FUNCTION_BLOCK FB_Axis
VAR_OUTPUT
	bError			:	BOOL;				//Error signal
	nErrorID		:	UDINT;				//Error ID
	bMoving			:	BOOL;				// Status of moving
END_VAR
VAR
	bResetDone		:	BOOL;				// Status of function block MC_Reset
	bHaltDone		:	BOOL;				// Status of function block MC_Halt

	bStatusEnable	:	BOOL;				// Enable feedback
	
	fVelocity		:	LREAL;				// Target velocity
	fOverride		:	LREAL := 100;		// Override 100%
	
	fbTriggerHalt	:	R_TRIG;				// Trigger to recognize rising edge of halt input
	fbTriggerReset	:	R_TRIG;				// Trigger to recognize rising edge of reset input
	
	AxisRef			:	AXIS_REF;			// Axis reference (process data plc/nc)
	
	//=============== Motion function blocks =====================
	fbMcPower		:	MC_Power;			// FB for enable and override
	fbMcReset		:	MC_Reset;			// FB to reset axis (errors)
	fbMcStop		:	MC_Stop;				// FB to stop axis
	fbMcHalt		:	MC_Halt;				// FB to halt axis
	fbMcMove		:	Mc_MoveVelocity;	// FB to move axis (velocity movement)
	fbMcMoveAbsolute :	Mc_MoveAbsolute;	// FB to move axis (absolute position)
END_VAR

PROPERTY bState_Enable : BOOL
GET
bState_Enable := bStatusEnable;
END_GET
END_PROPERTY

PROPERTY bState_HaltDone : BOOL
GET
bState_HaltDone := bHaltDone;
END_GET
END_PROPERTY

PROPERTY bState_ResetDone : BOOL
GET
bState_ResetDone := bResetDone;
END_GET
END_PROPERTY

METHOD Enable
VAR_INPUT
	bEnable		:		BOOL;
END_VAR
fbMcPower(	Axis 			:= THIS^.AxisRef,
			Enable 			:=  bEnable,
			Enable_Positive := bEnable,
			Enable_Negative := bEnable,
			Override 		:= THIS^.fOverride,
			Status 			=> THIS^.bStatusEnable);
			
IF fbMcPower.Error THEN
	bError		:= TRUE;
	nErrorID	:= fbMcPower.ErrorID;
END_IF

AxisRef.ReadStatus();		// Axis internal method to read its status

THIS^.bMoving := AxisRef.Status.Moving;
END_METHOD

PROPERTY fTargetVelocity : LREAL
GET
fTargetVelocity := fVelocity;
END_GET
SET
fVelocity := fTargetVelocity;
END_SET
END_PROPERTY

METHOD Halt
VAR_INPUT
	bDriveHalt	:	BOOL;
END_VAR
// Move axis command set to FALSE
IF bDriveHalt THEN
	THIS^.fbMcMove( Axis 				:= THIS^.AxisRef,
					Execute 			:= FALSE);
	// ?? Move Absolute Execute FALSE ??
	THIS^.fbMcMoveAbsolute( Axis 		:= THIS^.AxisRef,
							Execute 	:= FALSE);		
ELSE
	THIS^.bHaltDone := FALSE;				
END_IF

//Trigger
THIS^.fbTriggerHalt(CLK := bDriveHalt);

IF THIS^.fbTriggerHalt.Q THEN
	THIS^.fbMcHalt( Axis			:= THIS^.AxisRef,
					Execute			:= TRUE);
ELSE
	THIS^.fbMcHalt( Axis			:= THIS^.AxisRef);
END_IF

// Done / Error / Aborted
IF THIS^.fbMcHalt.Done OR THIS^.fbMcHalt.Error OR THIS^.fbMcHalt.CommandAborted THEN
	THIS^.bError		:= THIS^.fbMcHalt.Error;
	THIS^.nErrorID		:= THIS^.fbMcHalt.ErrorID;
	THIS^.bHaltDone		:= THIS^.fbMcHalt.Done;

	THIS^.fbMcHalt( Axis 		:= THIS^.AxisRef,
					Execute		:= FALSE);
END_IF
END_METHOD

METHOD MoveBw
VAR_INPUT
END_VAR
IF NOT THIS^.fbMcMove.Error THEN
	fbMcMove(	Axis		:= THIS^.AxisRef,
				Execute		:= TRUE,
				Direction	:= MC_Negative_Direction,
				Velocity	:= THIS^.fVelocity);
END_IF

// Error / Command aborted
IF THIS^.fbMcMove.Error OR THIS^.fbMcMove.CommandAborted THEN
	THIS^.bError			:= THIS^.fbMcMove.Error;
	THIS^.nErrorID			:= THIS^.fbMcMove.ErrorID;
END_IF

	fbMcMove(	Axis		:= THIS^.AxisRef,
				Execute		:= FALSE);
END_METHOD

METHOD MoveFw
VAR_INPUT
END_VAR
IF NOT THIS^.fbMcMove.Error THEN
	fbMcMove(	Axis		:= THIS^.AxisRef,
				Execute		:= TRUE,
				Direction	:= MC_Positive_Direction,
				Velocity	:= THIS^.fVelocity);
END_IF

// Error / Command aborted
IF THIS^.fbMcMove.Error OR THIS^.fbMcMove.CommandAborted THEN
	THIS^.bError			:= THIS^.fbMcMove.Error;
	THIS^.nErrorID			:= THIS^.fbMcMove.ErrorID;
END_IF

	fbMcMove(	Axis		:= THIS^.AxisRef,
				Execute		:= FALSE);
END_METHOD

METHOD Reset
VAR_INPUT
	bDriveReset		:	BOOL;	// Request reset
END_VAR
IF NOT bDriveReset THEN
	THIS^.bResetDone := FALSE;
END_IF

// Trigger
THIS^.fbTriggerReset(CLK 		:= bDriveReset);

IF THIS^.fbTriggerReset.Q THEN
	THIS^.bResetDone := FALSE;
	THIS^.fbMcReset(Axis 		:= THIS^.AxisRef,
					Execute 	:= TRUE);
ELSE
	THIS^.fbMcReset(Axis 		:= THIS^.AxisRef);
END_IF

// Done / Error
IF THIS^.fbMcReset.Done OR THIS^.fbMcReset.Error THEN
	THIS^.bResetDone 			:= THIS^.fbMcReset.Done;
	THIS^.bError		 		:= THIS^.fbMcReset.Error;
	
	THIS^.fbMcReset (Axis 		:= THIS^.AxisRef,
					Execute 	:= FALSE);
END_IF
END_METHOD

METHOD Stop
VAR_INPUT
	bDriveStop	:	BOOL;		// Request drive stop
END_VAR
IF bDriveStop THEN
	// Move Execute FALSE
	THIS^.fbMcMove( Axis 				:= THIS^.AxisRef,
					Execute 			:= FALSE);			
	// ?? Move Absolute Execute FALSE ??
	THIS^.fbMcMoveAbsolute( Axis 		:= THIS^.AxisRef,
							Execute 	:= FALSE);			

ELSE
	THIS^.bHaltDone := FALSE;
END_IF

// Trigger
THIS^.fbTriggerHalt(CLK := bDriveStop);

IF fbTriggerHalt.Q THEN
	THIS^.fbMcStop( Axis 		:= THIS^.AxisRef,
					Execute 	:= TRUE);
END_IF

// Done / Error / Command aborted
IF THIS^.fbMcStop.Done OR THIS^.fbMcStop.Error OR THIS^.fbMcStop.CommandAborted THEN
	THIS^.bError				:= THIS^.fbMcStop.Error;
	THIS^.bError				:= THIS^.fbMcStop.Error;
	THIS^.bHaltDone				:= THIS^.fbMcStop.Done;
	
	THIS^.fbMcStop( Axis 		:= THIS^.AxisRef,
					Execute 	:= FALSE);
	
END_IF
END_METHOD

END_FUNCTION_BLOCK

(* stored: Version 1.1.0.1, ProductVersion 3.1.4024.15
   POU FB_Axis: Id {6c8846af-ad09-42ea-ac30-58778bca0d31}, SpecialFunc None
   Property bState_Enable: Id {cd309e48-5f46-43f7-8c5f-38c97dbe91a3}
   Get Get: Id {44efe57e-5c77-4d97-a9f5-87e818569938}
   Property bState_HaltDone: Id {d8afc25b-a64c-4b9f-83bf-134bde42221b}
   Get Get: Id {f9e3e88c-d7b9-441d-b557-bad23cd20934}
   Property bState_ResetDone: Id {4c75998b-c40e-4509-80ad-9daefe9db7c9}
   Get Get: Id {c50b97b6-3014-48f3-88f6-bbfa1ae68ccc}
   Method Enable: Id {11193f3f-f540-4489-a639-5127b8d49d56}
   Property fTargetVelocity: Id {652d5236-2979-48da-a9f1-d13a0a90f62f}
   Get Get: Id {b936ae19-6acb-4c8d-9ec0-2a49bb0e0b26}
   Set Set: Id {f58b27e8-4200-4ceb-8453-506e7d075242}
   Method Halt: Id {f9112d11-079e-466e-84db-189b8da28e33}
   Method MoveBw: Id {a783e9b0-c4cb-42e5-9e17-a4b39013e7dc}
   Method MoveFw: Id {85439bc6-9d48-4242-b8ca-4942cbad842a}
   Method Reset: Id {e170a953-3cb8-44ac-a18c-770eddd0d1c2}
   Method Stop: Id {8a05423b-97ae-4aab-ad6a-e9217e3f8502} *)
